PROGRAM F14_CaseQueueControl
VAR_OUTPUT
END_VAR
VAR
	fbInterPushCaseQueueIndex			: FB_CASE_ShiftCaseQueue;
	fbCaseCompleteCaseQueueIndex		: FB_CASE_ShiftCaseQueue;
	fbCaseDiscargeQueueMove			: FB_CASE_ShiftCaseQueue;

	srDischargeIndexing					: SR;
	srWaitingToScanCaseLabel			: SR;

	rtrigCaseDischarge				: R_TRIG;
	rtrigCaseComplete				: R_TRIG;
	rtrigCaseWaitingToScanLabel		: R_TRIG;

END_VAR

(*
Modification history:
Date		|	Author 		|	Remark
----------------------------------------------------------------------------------------------------
02.09.20	|	PP			|	Start Remarking.
*)

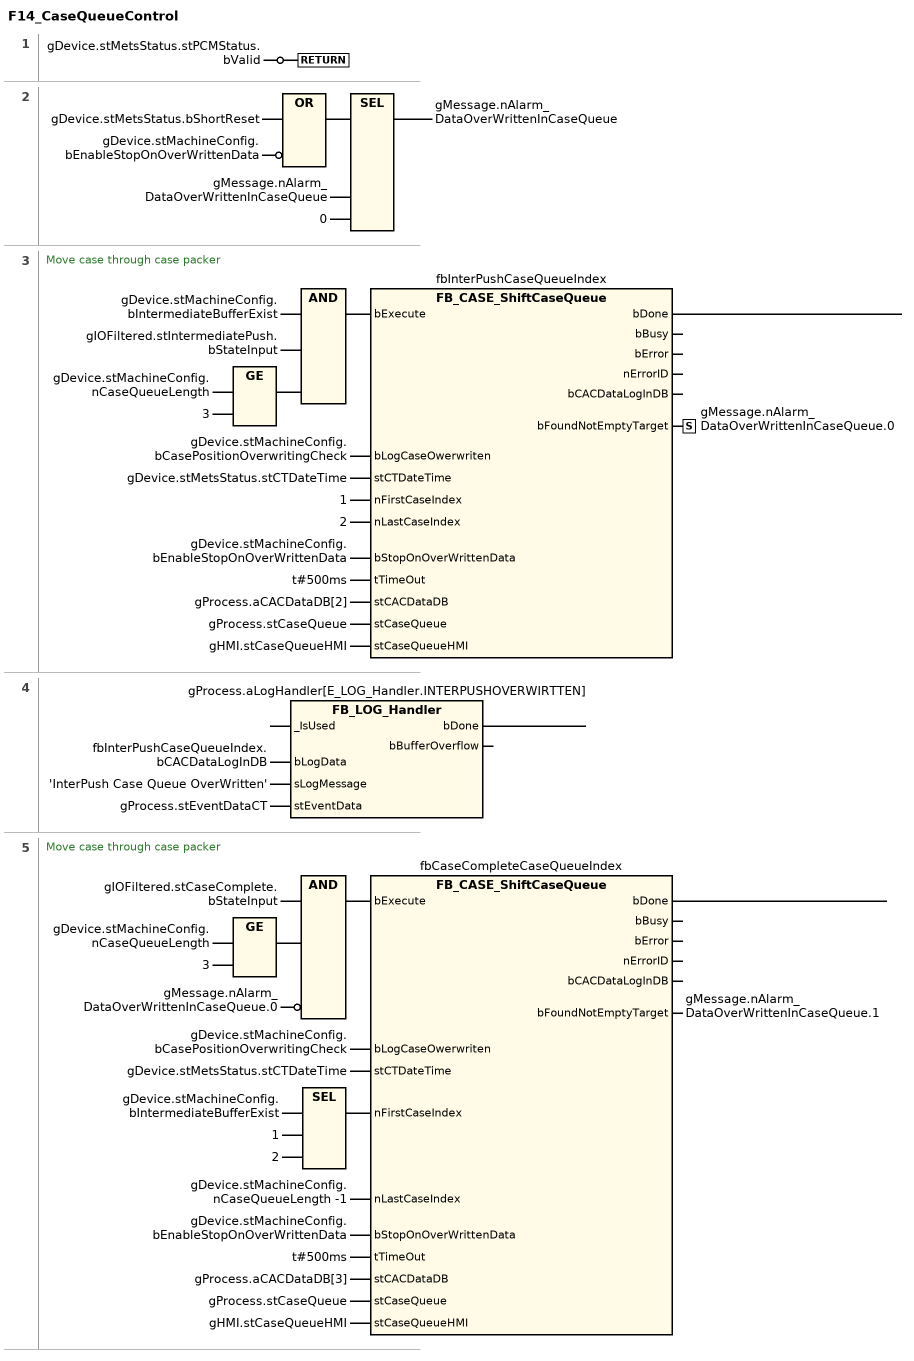
// NETWORK 1
IF NOT gDevice.stMetsStatus.stPCMStatus.bValid THEN RETURN; END_IF

// NETWORK 2
gMessage.nAlarm_DataOverWrittenInCaseQueue := SEL(gDevice.stMetsStatus.bShortReset OR NOT gDevice.stMachineConfig.bEnableStopOnOverWrittenData, gMessage.nAlarm_DataOverWrittenInCaseQueue, 0);

// NETWORK 3
// Move case through case packer
fbInterPushCaseQueueIndex(
    bExecute := gDevice.stMachineConfig.bIntermediateBufferExist AND gIOFiltered.stIntermediatePush.bStateInput AND gDevice.stMachineConfig.nCaseQueueLength >= 3,
    bLogCaseOwerwriten := gDevice.stMachineConfig.bCasePositionOverwritingCheck,
    stCTDateTime := gDevice.stMetsStatus.stCTDateTime,
    nFirstCaseIndex := 1,
    nLastCaseIndex := 2,
    bStopOnOverWrittenData := gDevice.stMachineConfig.bEnableStopOnOverWrittenData,
    tTimeOut := t#500ms,
    stCACDataDB := gProcess.aCACDataDB[2],
    stCaseQueue := gProcess.stCaseQueue,
    stCaseQueueHMI := gHMI.stCaseQueueHMI); // FB_CASE_ShiftCaseQueue
gMessage.nAlarm_DataOverWrittenInCaseQueue.0 S= fbInterPushCaseQueueIndex.bFoundNotEmptyTarget;

// NETWORK 4
gProcess.aLogHandler[E_LOG_Handler.INTERPUSHOVERWIRTTEN](
    bLogData := fbInterPushCaseQueueIndex.bCACDataLogInDB,
    sLogMessage := 'InterPush Case Queue OverWritten',
    stEventData := gProcess.stEventDataCT); // FB_LOG_Handler

// NETWORK 5
// Move case through case packer
fbCaseCompleteCaseQueueIndex(
    bExecute := gIOFiltered.stCaseComplete.bStateInput AND gDevice.stMachineConfig.nCaseQueueLength >= 3 AND NOT gMessage.nAlarm_DataOverWrittenInCaseQueue.0,
    bLogCaseOwerwriten := gDevice.stMachineConfig.bCasePositionOverwritingCheck,
    stCTDateTime := gDevice.stMetsStatus.stCTDateTime,
    nFirstCaseIndex := SEL(gDevice.stMachineConfig.bIntermediateBufferExist, 1, 2),
    nLastCaseIndex := gDevice.stMachineConfig.nCaseQueueLength -1,
    bStopOnOverWrittenData := gDevice.stMachineConfig.bEnableStopOnOverWrittenData,
    tTimeOut := t#500ms,
    stCACDataDB := gProcess.aCACDataDB[3],
    stCaseQueue := gProcess.stCaseQueue,
    stCaseQueueHMI := gHMI.stCaseQueueHMI,
    bFoundNotEmptyTarget => gMessage.nAlarm_DataOverWrittenInCaseQueue.1); // FB_CASE_ShiftCaseQueue

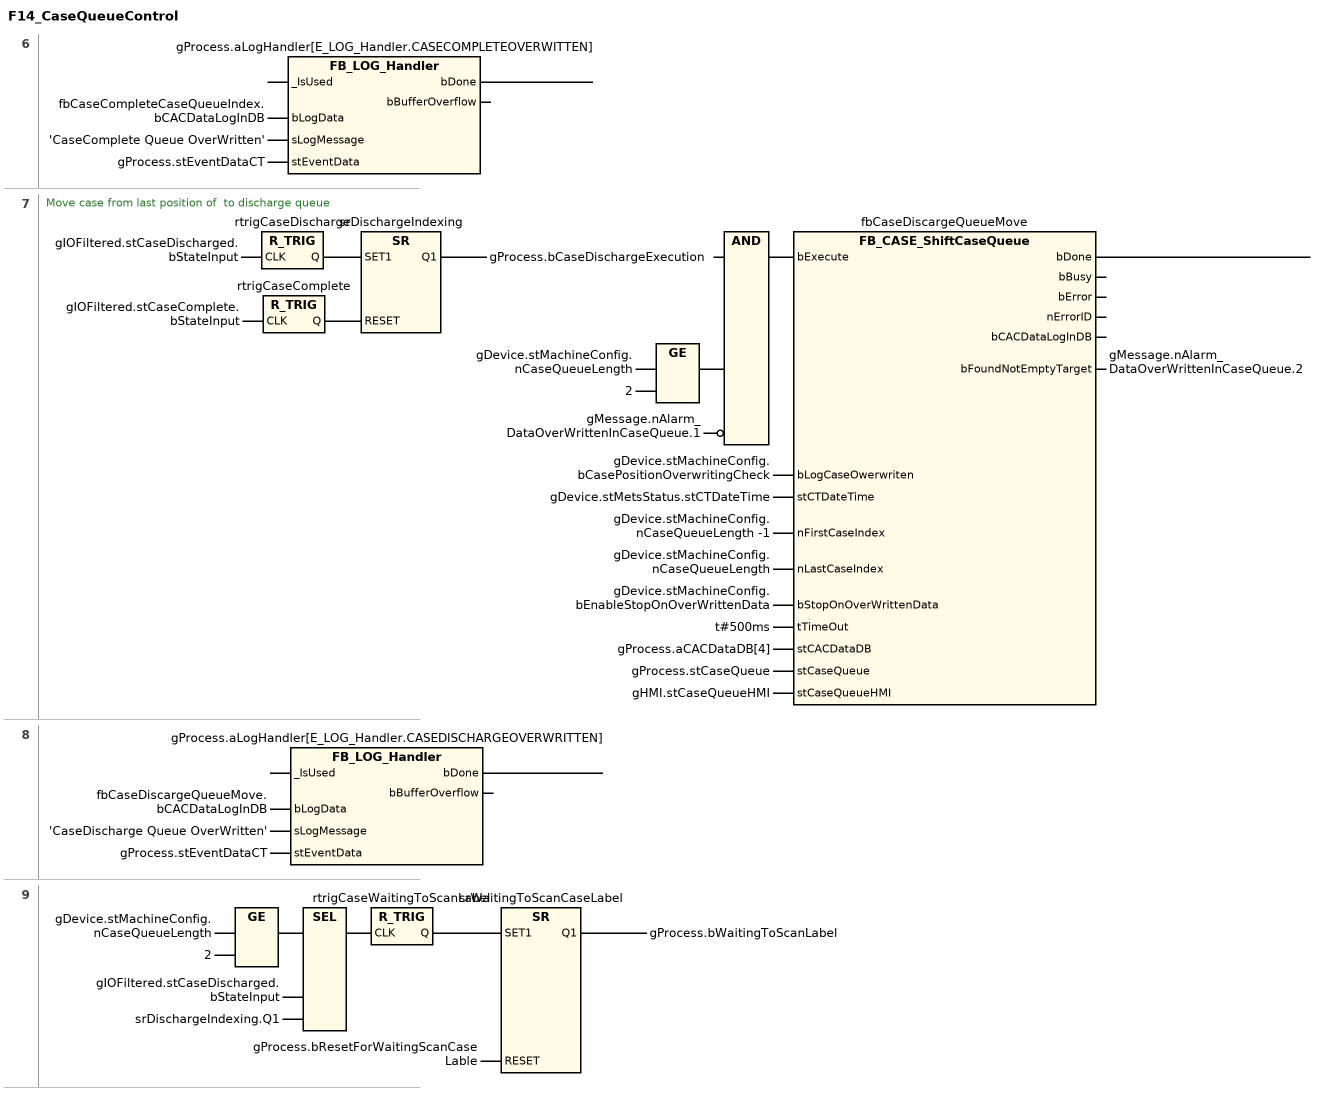
// NETWORK 6
gProcess.aLogHandler[E_LOG_Handler.CASECOMPLETEOVERWITTEN](
    bLogData := fbCaseCompleteCaseQueueIndex.bCACDataLogInDB,
    sLogMessage := 'CaseComplete Queue OverWritten',
    stEventData := gProcess.stEventDataCT); // FB_LOG_Handler

// NETWORK 7
// Move case from last position of  to discharge queue
rtrigCaseDischarge(CLK := gIOFiltered.stCaseDischarged.bStateInput); // R_TRIG
rtrigCaseComplete(CLK := gIOFiltered.stCaseComplete.bStateInput); // R_TRIG
srDischargeIndexing(SET1 := rtrigCaseDischarge.Q, RESET := rtrigCaseComplete.Q); // SR
gProcess.bCaseDischargeExecution := srDischargeIndexing.Q1;
fbCaseDiscargeQueueMove(
    bExecute := srDischargeIndexing.Q1 AND gDevice.stMachineConfig.nCaseQueueLength >= 2 AND NOT gMessage.nAlarm_DataOverWrittenInCaseQueue.1,
    bLogCaseOwerwriten := gDevice.stMachineConfig.bCasePositionOverwritingCheck,
    stCTDateTime := gDevice.stMetsStatus.stCTDateTime,
    nFirstCaseIndex := gDevice.stMachineConfig.nCaseQueueLength -1,
    nLastCaseIndex := gDevice.stMachineConfig.nCaseQueueLength,
    bStopOnOverWrittenData := gDevice.stMachineConfig.bEnableStopOnOverWrittenData,
    tTimeOut := t#500ms,
    stCACDataDB := gProcess.aCACDataDB[4],
    stCaseQueue := gProcess.stCaseQueue,
    stCaseQueueHMI := gHMI.stCaseQueueHMI,
    bFoundNotEmptyTarget => gMessage.nAlarm_DataOverWrittenInCaseQueue.2); // FB_CASE_ShiftCaseQueue

// NETWORK 8
gProcess.aLogHandler[E_LOG_Handler.CASEDISCHARGEOVERWRITTEN](
    bLogData := fbCaseDiscargeQueueMove.bCACDataLogInDB,
    sLogMessage := 'CaseDischarge Queue OverWritten',
    stEventData := gProcess.stEventDataCT); // FB_LOG_Handler

// NETWORK 9
rtrigCaseWaitingToScanLabel(CLK := SEL(gDevice.stMachineConfig.nCaseQueueLength >= 2, gIOFiltered.stCaseDischarged.bStateInput, srDischargeIndexing.Q1)); // R_TRIG
srWaitingToScanCaseLabel(SET1 := rtrigCaseWaitingToScanLabel.Q, RESET := gProcess.bResetForWaitingScanCaseLable); // SR
gProcess.bWaitingToScanLabel := srWaitingToScanCaseLabel.Q1;

END_PROGRAM

(* stored: Version 1.1.0.1
   POU F14_CaseQueueControl: Id {fe0cc1c3-7044-4c3c-9c14-7560f8e5bb84}, SpecialFunc None *)
